// TIA Portal V19 export
FUNCTION "SUBOUTPUT" : Void   // FC4, LAD
{ S7_Optimized_Access := 'TRUE' }
// stored: SetENOAutomatically false
BEGIN

REGION Network 1: P-202 A RO 1 FEED PUMP
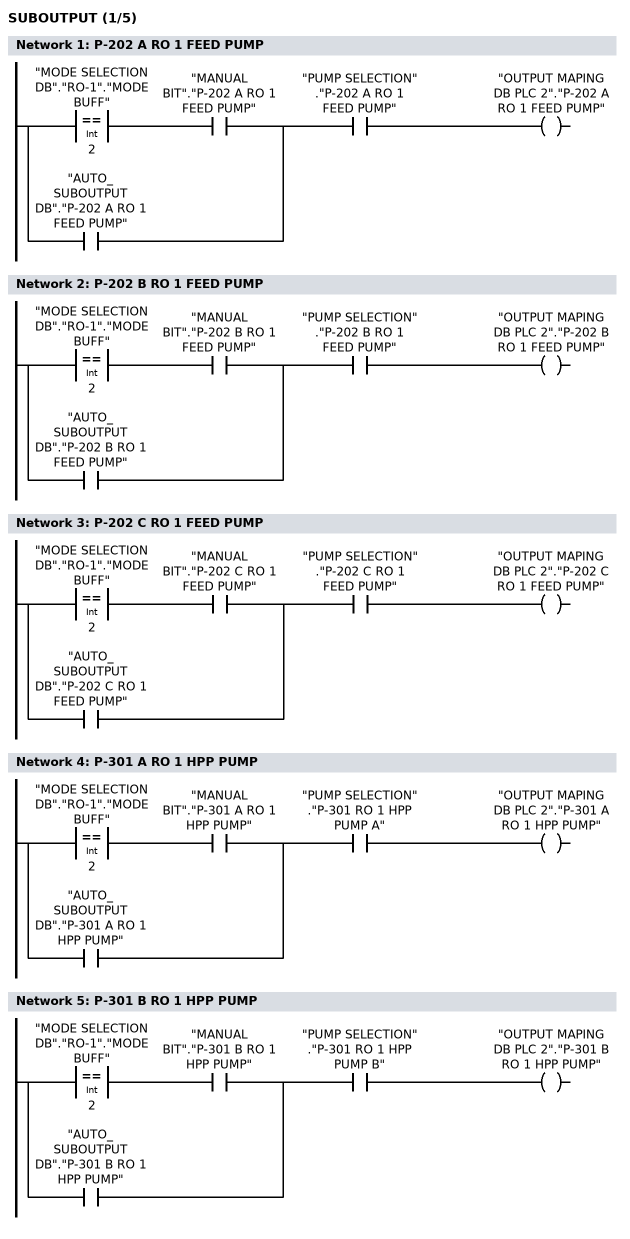
   RUNG wire#powerrail
      { S7_Templates := "SrcType := Int" } EQ_Contact(in1 := "MODE SELECTION DB"."RO-1"."MODE BUFF", in2 := 2)
      Contact( "MANUAL BIT"."P-202 A RO 1 FEED PUMP" )
      wire#w1
      Contact( "PUMP SELECTION"."P-202 A RO 1 FEED PUMP" )
      Coil( "OUTPUT MAPING DB PLC 2"."P-202 A RO 1 FEED PUMP" )
   END_RUNG
   RUNG wire#powerrail
      Contact( "AUTO_SUBOUTPUT DB"."P-202 A RO 1 FEED PUMP" )
   END_RUNG wire#w1
   // the same network as SCL:
   "OUTPUT MAPING DB PLC 2"."P-202 A RO 1 FEED PUMP" := ((("MODE SELECTION DB"."RO-1"."MODE BUFF" = 2) AND "MANUAL BIT"."P-202 A RO 1 FEED PUMP") OR "AUTO_SUBOUTPUT DB"."P-202 A RO 1 FEED PUMP") AND "PUMP SELECTION"."P-202 A RO 1 FEED PUMP";
END_REGION

REGION Network 2: P-202 B RO 1 FEED PUMP
   RUNG wire#powerrail
      { S7_Templates := "SrcType := Int" } EQ_Contact(in1 := "MODE SELECTION DB"."RO-1"."MODE BUFF", in2 := 2)
      Contact( "MANUAL BIT"."P-202 B RO 1 FEED PUMP" )
      wire#w1
      Contact( "PUMP SELECTION"."P-202 B RO 1 FEED PUMP" )
      Coil( "OUTPUT MAPING DB PLC 2"."P-202 B RO 1 FEED PUMP" )
   END_RUNG
   RUNG wire#powerrail
      Contact( "AUTO_SUBOUTPUT DB"."P-202 B RO 1 FEED PUMP" )
   END_RUNG wire#w1
   // the same network as SCL:
   "OUTPUT MAPING DB PLC 2"."P-202 B RO 1 FEED PUMP" := ((("MODE SELECTION DB"."RO-1"."MODE BUFF" = 2) AND "MANUAL BIT"."P-202 B RO 1 FEED PUMP") OR "AUTO_SUBOUTPUT DB"."P-202 B RO 1 FEED PUMP") AND "PUMP SELECTION"."P-202 B RO 1 FEED PUMP";
END_REGION

REGION Network 3: P-202 C RO 1 FEED PUMP
   RUNG wire#powerrail
      { S7_Templates := "SrcType := Int" } EQ_Contact(in1 := "MODE SELECTION DB"."RO-1"."MODE BUFF", in2 := 2)
      Contact( "MANUAL BIT"."P-202 C RO 1 FEED PUMP" )
      wire#w1
      Contact( "PUMP SELECTION"."P-202 C RO 1 FEED PUMP" )
      Coil( "OUTPUT MAPING DB PLC 2"."P-202 C RO 1 FEED PUMP" )
   END_RUNG
   RUNG wire#powerrail
      Contact( "AUTO_SUBOUTPUT DB"."P-202 C RO 1 FEED PUMP" )
   END_RUNG wire#w1
   // the same network as SCL:
   "OUTPUT MAPING DB PLC 2"."P-202 C RO 1 FEED PUMP" := ((("MODE SELECTION DB"."RO-1"."MODE BUFF" = 2) AND "MANUAL BIT"."P-202 C RO 1 FEED PUMP") OR "AUTO_SUBOUTPUT DB"."P-202 C RO 1 FEED PUMP") AND "PUMP SELECTION"."P-202 C RO 1 FEED PUMP";
END_REGION

REGION Network 4: P-301 A RO 1 HPP PUMP
   RUNG wire#powerrail
      { S7_Templates := "SrcType := Int" } EQ_Contact(in1 := "MODE SELECTION DB"."RO-1"."MODE BUFF", in2 := 2)
      Contact( "MANUAL BIT"."P-301 A RO 1 HPP PUMP" )
      wire#w1
      Contact( "PUMP SELECTION"."P-301 RO 1 HPP PUMP A" )
      Coil( "OUTPUT MAPING DB PLC 2"."P-301 A RO 1 HPP PUMP" )
   END_RUNG
   RUNG wire#powerrail
      Contact( "AUTO_SUBOUTPUT DB"."P-301 A RO 1 HPP PUMP" )
   END_RUNG wire#w1
   // the same network as SCL:
   "OUTPUT MAPING DB PLC 2"."P-301 A RO 1 HPP PUMP" := ((("MODE SELECTION DB"."RO-1"."MODE BUFF" = 2) AND "MANUAL BIT"."P-301 A RO 1 HPP PUMP") OR "AUTO_SUBOUTPUT DB"."P-301 A RO 1 HPP PUMP") AND "PUMP SELECTION"."P-301 RO 1 HPP PUMP A";
END_REGION

REGION Network 5: P-301 B RO 1 HPP PUMP
   RUNG wire#powerrail
      { S7_Templates := "SrcType := Int" } EQ_Contact(in1 := "MODE SELECTION DB"."RO-1"."MODE BUFF", in2 := 2)
      Contact( "MANUAL BIT"."P-301 B RO 1 HPP PUMP" )
      wire#w1
      Contact( "PUMP SELECTION"."P-301 RO 1 HPP PUMP B" )
      Coil( "OUTPUT MAPING DB PLC 2"."P-301 B RO 1 HPP PUMP" )
   END_RUNG
   RUNG wire#powerrail
      Contact( "AUTO_SUBOUTPUT DB"."P-301 B RO 1 HPP PUMP" )
   END_RUNG wire#w1
   // the same network as SCL:
   "OUTPUT MAPING DB PLC 2"."P-301 B RO 1 HPP PUMP" := ((("MODE SELECTION DB"."RO-1"."MODE BUFF" = 2) AND "MANUAL BIT"."P-301 B RO 1 HPP PUMP") OR "AUTO_SUBOUTPUT DB"."P-301 B RO 1 HPP PUMP") AND "PUMP SELECTION"."P-301 RO 1 HPP PUMP B";
END_REGION

REGION Network 6: P-401 A RO 2 FEED PUMP
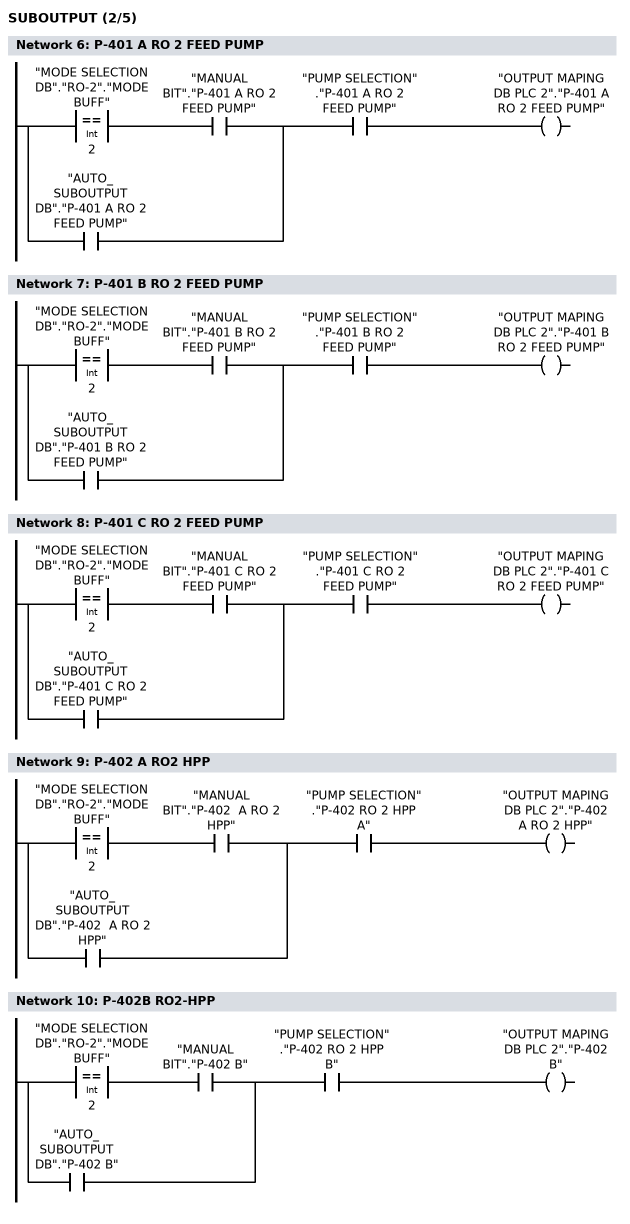
   RUNG wire#powerrail
      { S7_Templates := "SrcType := Int" } EQ_Contact(in1 := "MODE SELECTION DB"."RO-2"."MODE BUFF", in2 := 2)
      Contact( "MANUAL BIT"."P-401 A RO 2 FEED PUMP" )
      wire#w1
      Contact( "PUMP SELECTION"."P-401 A RO 2 FEED PUMP" )
      Coil( "OUTPUT MAPING DB PLC 2"."P-401 A RO 2 FEED PUMP" )
   END_RUNG
   RUNG wire#powerrail
      Contact( "AUTO_SUBOUTPUT DB"."P-401 A RO 2 FEED PUMP" )
   END_RUNG wire#w1
   // the same network as SCL:
   "OUTPUT MAPING DB PLC 2"."P-401 A RO 2 FEED PUMP" := ((("MODE SELECTION DB"."RO-2"."MODE BUFF" = 2) AND "MANUAL BIT"."P-401 A RO 2 FEED PUMP") OR "AUTO_SUBOUTPUT DB"."P-401 A RO 2 FEED PUMP") AND "PUMP SELECTION"."P-401 A RO 2 FEED PUMP";
END_REGION

REGION Network 7: P-401 B RO 2 FEED PUMP
   RUNG wire#powerrail
      { S7_Templates := "SrcType := Int" } EQ_Contact(in1 := "MODE SELECTION DB"."RO-2"."MODE BUFF", in2 := 2)
      Contact( "MANUAL BIT"."P-401 B RO 2 FEED PUMP" )
      wire#w1
      Contact( "PUMP SELECTION"."P-401 B RO 2 FEED PUMP" )
      Coil( "OUTPUT MAPING DB PLC 2"."P-401 B RO 2 FEED PUMP" )
   END_RUNG
   RUNG wire#powerrail
      Contact( "AUTO_SUBOUTPUT DB"."P-401 B RO 2 FEED PUMP" )
   END_RUNG wire#w1
   // the same network as SCL:
   "OUTPUT MAPING DB PLC 2"."P-401 B RO 2 FEED PUMP" := ((("MODE SELECTION DB"."RO-2"."MODE BUFF" = 2) AND "MANUAL BIT"."P-401 B RO 2 FEED PUMP") OR "AUTO_SUBOUTPUT DB"."P-401 B RO 2 FEED PUMP") AND "PUMP SELECTION"."P-401 B RO 2 FEED PUMP";
END_REGION

REGION Network 8: P-401 C RO 2 FEED PUMP
   RUNG wire#powerrail
      { S7_Templates := "SrcType := Int" } EQ_Contact(in1 := "MODE SELECTION DB"."RO-2"."MODE BUFF", in2 := 2)
      Contact( "MANUAL BIT"."P-401 C RO 2 FEED PUMP" )
      wire#w1
      Contact( "PUMP SELECTION"."P-401 C RO 2 FEED PUMP" )
      Coil( "OUTPUT MAPING DB PLC 2"."P-401 C RO 2 FEED PUMP" )
   END_RUNG
   RUNG wire#powerrail
      Contact( "AUTO_SUBOUTPUT DB"."P-401 C RO 2 FEED PUMP" )
   END_RUNG wire#w1
   // the same network as SCL:
   "OUTPUT MAPING DB PLC 2"."P-401 C RO 2 FEED PUMP" := ((("MODE SELECTION DB"."RO-2"."MODE BUFF" = 2) AND "MANUAL BIT"."P-401 C RO 2 FEED PUMP") OR "AUTO_SUBOUTPUT DB"."P-401 C RO 2 FEED PUMP") AND "PUMP SELECTION"."P-401 C RO 2 FEED PUMP";
END_REGION

REGION Network 9: P-402 A RO2 HPP
   RUNG wire#powerrail
      { S7_Templates := "SrcType := Int" } EQ_Contact(in1 := "MODE SELECTION DB"."RO-2"."MODE BUFF", in2 := 2)
      Contact( "MANUAL BIT"."P-402  A RO 2 HPP" )
      wire#w1
      Contact( "PUMP SELECTION"."P-402 RO 2 HPP A" )
      Coil( "OUTPUT MAPING DB PLC 2"."P-402  A RO 2 HPP" )
   END_RUNG
   RUNG wire#powerrail
      Contact( "AUTO_SUBOUTPUT DB"."P-402  A RO 2 HPP" )
   END_RUNG wire#w1
   // the same network as SCL:
   "OUTPUT MAPING DB PLC 2"."P-402  A RO 2 HPP" := ((("MODE SELECTION DB"."RO-2"."MODE BUFF" = 2) AND "MANUAL BIT"."P-402  A RO 2 HPP") OR "AUTO_SUBOUTPUT DB"."P-402  A RO 2 HPP") AND "PUMP SELECTION"."P-402 RO 2 HPP A";
END_REGION

REGION Network 10: P-402B RO2-HPP
   RUNG wire#powerrail
      { S7_Templates := "SrcType := Int" } EQ_Contact(in1 := "MODE SELECTION DB"."RO-2"."MODE BUFF", in2 := 2)
      Contact( "MANUAL BIT"."P-402 B" )
      wire#w1
      Contact( "PUMP SELECTION"."P-402 RO 2 HPP B" )
      Coil( "OUTPUT MAPING DB PLC 2"."P-402 B" )
   END_RUNG
   RUNG wire#powerrail
      Contact( "AUTO_SUBOUTPUT DB"."P-402 B" )
   END_RUNG wire#w1
   // the same network as SCL:
   "OUTPUT MAPING DB PLC 2"."P-402 B" := ((("MODE SELECTION DB"."RO-2"."MODE BUFF" = 2) AND "MANUAL BIT"."P-402 B") OR "AUTO_SUBOUTPUT DB"."P-402 B") AND "PUMP SELECTION"."P-402 RO 2 HPP B";
END_REGION

REGION Network 11: P-501 A EDI FEED PUMP
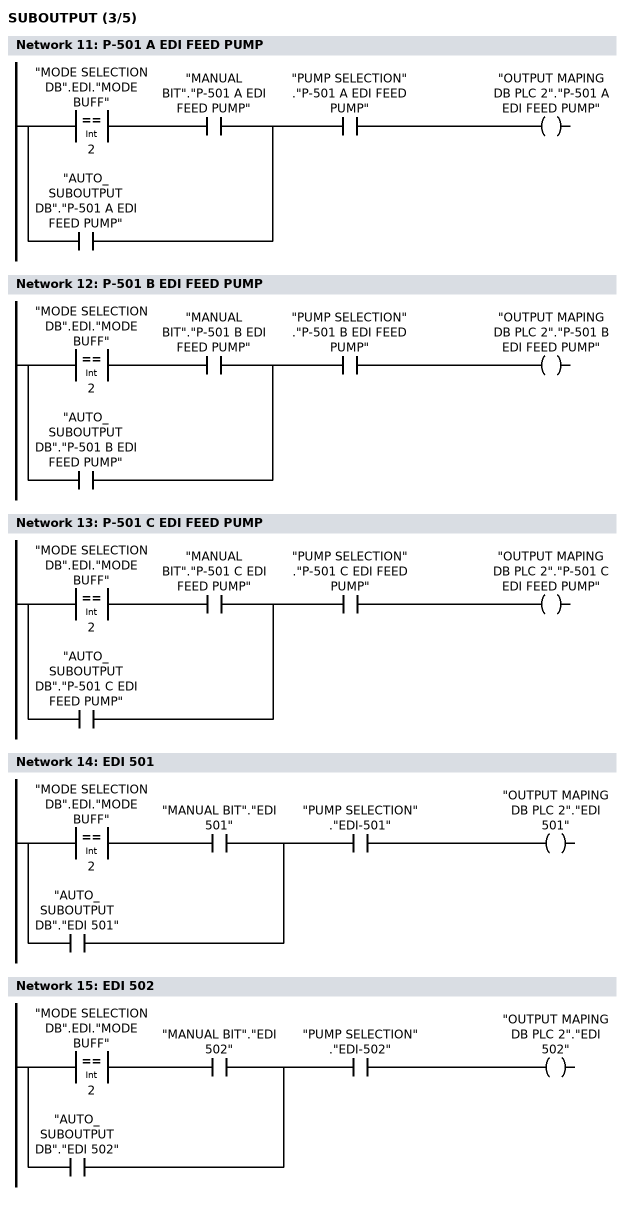
   RUNG wire#powerrail
      { S7_Templates := "SrcType := Int" } EQ_Contact(in1 := "MODE SELECTION DB".EDI."MODE BUFF", in2 := 2)
      Contact( "MANUAL BIT"."P-501 A EDI FEED PUMP" )
      wire#w1
      Contact( "PUMP SELECTION"."P-501 A EDI FEED PUMP" )
      Coil( "OUTPUT MAPING DB PLC 2"."P-501 A EDI FEED PUMP" )
   END_RUNG
   RUNG wire#powerrail
      Contact( "AUTO_SUBOUTPUT DB"."P-501 A EDI FEED PUMP" )
   END_RUNG wire#w1
   // the same network as SCL:
   "OUTPUT MAPING DB PLC 2"."P-501 A EDI FEED PUMP" := ((("MODE SELECTION DB".EDI."MODE BUFF" = 2) AND "MANUAL BIT"."P-501 A EDI FEED PUMP") OR "AUTO_SUBOUTPUT DB"."P-501 A EDI FEED PUMP") AND "PUMP SELECTION"."P-501 A EDI FEED PUMP";
END_REGION

REGION Network 12: P-501 B EDI FEED PUMP
   RUNG wire#powerrail
      { S7_Templates := "SrcType := Int" } EQ_Contact(in1 := "MODE SELECTION DB".EDI."MODE BUFF", in2 := 2)
      Contact( "MANUAL BIT"."P-501 B EDI FEED PUMP" )
      wire#w1
      Contact( "PUMP SELECTION"."P-501 B EDI FEED PUMP" )
      Coil( "OUTPUT MAPING DB PLC 2"."P-501 B EDI FEED PUMP" )
   END_RUNG
   RUNG wire#powerrail
      Contact( "AUTO_SUBOUTPUT DB"."P-501 B EDI FEED PUMP" )
   END_RUNG wire#w1
   // the same network as SCL:
   "OUTPUT MAPING DB PLC 2"."P-501 B EDI FEED PUMP" := ((("MODE SELECTION DB".EDI."MODE BUFF" = 2) AND "MANUAL BIT"."P-501 B EDI FEED PUMP") OR "AUTO_SUBOUTPUT DB"."P-501 B EDI FEED PUMP") AND "PUMP SELECTION"."P-501 B EDI FEED PUMP";
END_REGION

REGION Network 13: P-501 C EDI FEED PUMP
   RUNG wire#powerrail
      { S7_Templates := "SrcType := Int" } EQ_Contact(in1 := "MODE SELECTION DB".EDI."MODE BUFF", in2 := 2)
      Contact( "MANUAL BIT"."P-501 C EDI FEED PUMP" )
      wire#w1
      Contact( "PUMP SELECTION"."P-501 C EDI FEED PUMP" )
      Coil( "OUTPUT MAPING DB PLC 2"."P-501 C EDI FEED PUMP" )
   END_RUNG
   RUNG wire#powerrail
      Contact( "AUTO_SUBOUTPUT DB"."P-501 C EDI FEED PUMP" )
   END_RUNG wire#w1
   // the same network as SCL:
   "OUTPUT MAPING DB PLC 2"."P-501 C EDI FEED PUMP" := ((("MODE SELECTION DB".EDI."MODE BUFF" = 2) AND "MANUAL BIT"."P-501 C EDI FEED PUMP") OR "AUTO_SUBOUTPUT DB"."P-501 C EDI FEED PUMP") AND "PUMP SELECTION"."P-501 C EDI FEED PUMP";
END_REGION

REGION Network 14: EDI 501
   RUNG wire#powerrail
      { S7_Templates := "SrcType := Int" } EQ_Contact(in1 := "MODE SELECTION DB".EDI."MODE BUFF", in2 := 2)
      Contact( "MANUAL BIT"."EDI 501" )
      wire#w1
      Contact( "PUMP SELECTION"."EDI-501" )
      Coil( "OUTPUT MAPING DB PLC 2"."EDI 501" )
   END_RUNG
   RUNG wire#powerrail
      Contact( "AUTO_SUBOUTPUT DB"."EDI 501" )
   END_RUNG wire#w1
   // the same network as SCL:
   "OUTPUT MAPING DB PLC 2"."EDI 501" := ((("MODE SELECTION DB".EDI."MODE BUFF" = 2) AND "MANUAL BIT"."EDI 501") OR "AUTO_SUBOUTPUT DB"."EDI 501") AND "PUMP SELECTION"."EDI-501";
END_REGION

REGION Network 15: EDI 502
   RUNG wire#powerrail
      { S7_Templates := "SrcType := Int" } EQ_Contact(in1 := "MODE SELECTION DB".EDI."MODE BUFF", in2 := 2)
      Contact( "MANUAL BIT"."EDI 502" )
      wire#w1
      Contact( "PUMP SELECTION"."EDI-502" )
      Coil( "OUTPUT MAPING DB PLC 2"."EDI 502" )
   END_RUNG
   RUNG wire#powerrail
      Contact( "AUTO_SUBOUTPUT DB"."EDI 502" )
   END_RUNG wire#w1
   // the same network as SCL:
   "OUTPUT MAPING DB PLC 2"."EDI 502" := ((("MODE SELECTION DB".EDI."MODE BUFF" = 2) AND "MANUAL BIT"."EDI 502") OR "AUTO_SUBOUTPUT DB"."EDI 502") AND "PUMP SELECTION"."EDI-502";
END_REGION

REGION Network 16: DP 703
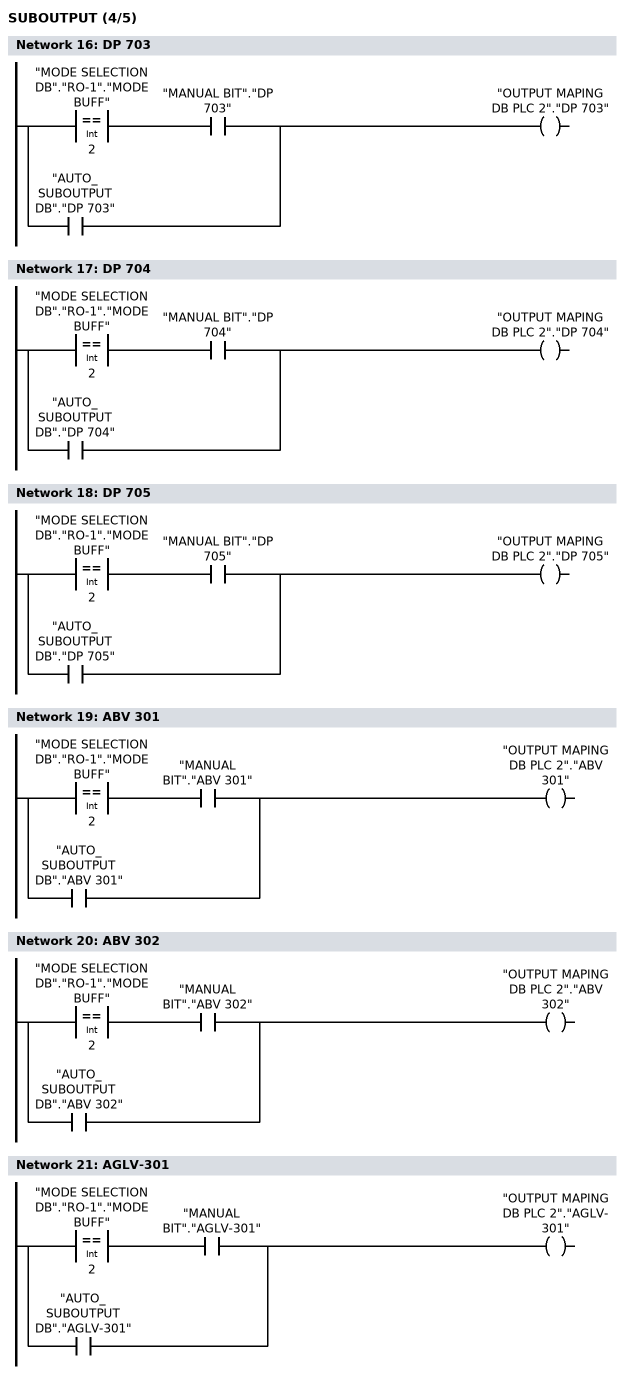
   RUNG wire#powerrail
      { S7_Templates := "SrcType := Int" } EQ_Contact(in1 := "MODE SELECTION DB"."RO-1"."MODE BUFF", in2 := 2)
      Contact( "MANUAL BIT"."DP 703" )
      wire#w1
      Coil( "OUTPUT MAPING DB PLC 2"."DP 703" )
   END_RUNG
   RUNG wire#powerrail
      Contact( "AUTO_SUBOUTPUT DB"."DP 703" )
   END_RUNG wire#w1
   // the same network as SCL:
   "OUTPUT MAPING DB PLC 2"."DP 703" := (("MODE SELECTION DB"."RO-1"."MODE BUFF" = 2) AND "MANUAL BIT"."DP 703") OR "AUTO_SUBOUTPUT DB"."DP 703";
END_REGION

REGION Network 17: DP 704
   RUNG wire#powerrail
      { S7_Templates := "SrcType := Int" } EQ_Contact(in1 := "MODE SELECTION DB"."RO-1"."MODE BUFF", in2 := 2)
      Contact( "MANUAL BIT"."DP 704" )
      wire#w1
      Coil( "OUTPUT MAPING DB PLC 2"."DP 704" )
   END_RUNG
   RUNG wire#powerrail
      Contact( "AUTO_SUBOUTPUT DB"."DP 704" )
   END_RUNG wire#w1
   // the same network as SCL:
   "OUTPUT MAPING DB PLC 2"."DP 704" := (("MODE SELECTION DB"."RO-1"."MODE BUFF" = 2) AND "MANUAL BIT"."DP 704") OR "AUTO_SUBOUTPUT DB"."DP 704";
END_REGION

REGION Network 18: DP 705
   RUNG wire#powerrail
      { S7_Templates := "SrcType := Int" } EQ_Contact(in1 := "MODE SELECTION DB"."RO-1"."MODE BUFF", in2 := 2)
      Contact( "MANUAL BIT"."DP 705" )
      wire#w1
      Coil( "OUTPUT MAPING DB PLC 2"."DP 705" )
   END_RUNG
   RUNG wire#powerrail
      Contact( "AUTO_SUBOUTPUT DB"."DP 705" )
   END_RUNG wire#w1
   // the same network as SCL:
   "OUTPUT MAPING DB PLC 2"."DP 705" := (("MODE SELECTION DB"."RO-1"."MODE BUFF" = 2) AND "MANUAL BIT"."DP 705") OR "AUTO_SUBOUTPUT DB"."DP 705";
END_REGION

REGION Network 19: ABV 301
   RUNG wire#powerrail
      { S7_Templates := "SrcType := Int" } EQ_Contact(in1 := "MODE SELECTION DB"."RO-1"."MODE BUFF", in2 := 2)
      Contact( "MANUAL BIT"."ABV 301" )
      wire#w1
      Coil( "OUTPUT MAPING DB PLC 2"."ABV 301" )
   END_RUNG
   RUNG wire#powerrail
      Contact( "AUTO_SUBOUTPUT DB"."ABV 301" )
   END_RUNG wire#w1
   // the same network as SCL:
   "OUTPUT MAPING DB PLC 2"."ABV 301" := (("MODE SELECTION DB"."RO-1"."MODE BUFF" = 2) AND "MANUAL BIT"."ABV 301") OR "AUTO_SUBOUTPUT DB"."ABV 301";
END_REGION

REGION Network 20: ABV 302
   RUNG wire#powerrail
      { S7_Templates := "SrcType := Int" } EQ_Contact(in1 := "MODE SELECTION DB"."RO-1"."MODE BUFF", in2 := 2)
      Contact( "MANUAL BIT"."ABV 302" )
      wire#w1
      Coil( "OUTPUT MAPING DB PLC 2"."ABV 302" )
   END_RUNG
   RUNG wire#powerrail
      Contact( "AUTO_SUBOUTPUT DB"."ABV 302" )
   END_RUNG wire#w1
   // the same network as SCL:
   "OUTPUT MAPING DB PLC 2"."ABV 302" := (("MODE SELECTION DB"."RO-1"."MODE BUFF" = 2) AND "MANUAL BIT"."ABV 302") OR "AUTO_SUBOUTPUT DB"."ABV 302";
END_REGION

REGION Network 21: AGLV-301
   RUNG wire#powerrail
      { S7_Templates := "SrcType := Int" } EQ_Contact(in1 := "MODE SELECTION DB"."RO-1"."MODE BUFF", in2 := 2)
      Contact( "MANUAL BIT"."AGLV-301" )
      wire#w1
      Coil( "OUTPUT MAPING DB PLC 2"."AGLV-301" )
   END_RUNG
   RUNG wire#powerrail
      Contact( "AUTO_SUBOUTPUT DB"."AGLV-301" )
   END_RUNG wire#w1
   // the same network as SCL:
   "OUTPUT MAPING DB PLC 2"."AGLV-301" := (("MODE SELECTION DB"."RO-1"."MODE BUFF" = 2) AND "MANUAL BIT"."AGLV-301") OR "AUTO_SUBOUTPUT DB"."AGLV-301";
END_REGION

REGION Network 22: AGLV-302
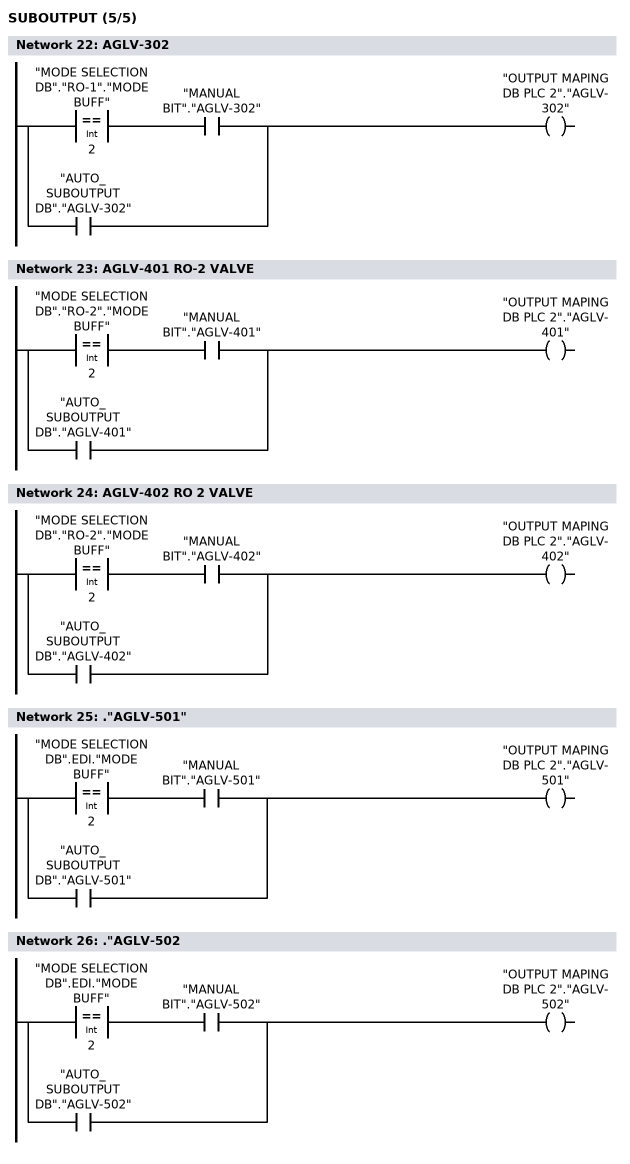
   RUNG wire#powerrail
      { S7_Templates := "SrcType := Int" } EQ_Contact(in1 := "MODE SELECTION DB"."RO-1"."MODE BUFF", in2 := 2)
      Contact( "MANUAL BIT"."AGLV-302" )
      wire#w1
      Coil( "OUTPUT MAPING DB PLC 2"."AGLV-302" )
   END_RUNG
   RUNG wire#powerrail
      Contact( "AUTO_SUBOUTPUT DB"."AGLV-302" )
   END_RUNG wire#w1
   // the same network as SCL:
   "OUTPUT MAPING DB PLC 2"."AGLV-302" := (("MODE SELECTION DB"."RO-1"."MODE BUFF" = 2) AND "MANUAL BIT"."AGLV-302") OR "AUTO_SUBOUTPUT DB"."AGLV-302";
END_REGION

REGION Network 23: AGLV-401 RO-2 VALVE
   RUNG wire#powerrail
      { S7_Templates := "SrcType := Int" } EQ_Contact(in1 := "MODE SELECTION DB"."RO-2"."MODE BUFF", in2 := 2)
      Contact( "MANUAL BIT"."AGLV-401" )
      wire#w1
      Coil( "OUTPUT MAPING DB PLC 2"."AGLV-401" )
   END_RUNG
   RUNG wire#powerrail
      Contact( "AUTO_SUBOUTPUT DB"."AGLV-401" )
   END_RUNG wire#w1
   // the same network as SCL:
   "OUTPUT MAPING DB PLC 2"."AGLV-401" := (("MODE SELECTION DB"."RO-2"."MODE BUFF" = 2) AND "MANUAL BIT"."AGLV-401") OR "AUTO_SUBOUTPUT DB"."AGLV-401";
END_REGION

REGION Network 24: AGLV-402 RO 2 VALVE
   RUNG wire#powerrail
      { S7_Templates := "SrcType := Int" } EQ_Contact(in1 := "MODE SELECTION DB"."RO-2"."MODE BUFF", in2 := 2)
      Contact( "MANUAL BIT"."AGLV-402" )
      wire#w1
      Coil( "OUTPUT MAPING DB PLC 2"."AGLV-402" )
   END_RUNG
   RUNG wire#powerrail
      Contact( "AUTO_SUBOUTPUT DB"."AGLV-402" )
   END_RUNG wire#w1
   // the same network as SCL:
   "OUTPUT MAPING DB PLC 2"."AGLV-402" := (("MODE SELECTION DB"."RO-2"."MODE BUFF" = 2) AND "MANUAL BIT"."AGLV-402") OR "AUTO_SUBOUTPUT DB"."AGLV-402";
END_REGION

REGION Network 25: ."AGLV-501"
   RUNG wire#powerrail
      { S7_Templates := "SrcType := Int" } EQ_Contact(in1 := "MODE SELECTION DB".EDI."MODE BUFF", in2 := 2)
      Contact( "MANUAL BIT"."AGLV-501" )
      wire#w1
      Coil( "OUTPUT MAPING DB PLC 2"."AGLV-501" )
   END_RUNG
   RUNG wire#powerrail
      Contact( "AUTO_SUBOUTPUT DB"."AGLV-501" )
   END_RUNG wire#w1
   // the same network as SCL:
   "OUTPUT MAPING DB PLC 2"."AGLV-501" := (("MODE SELECTION DB".EDI."MODE BUFF" = 2) AND "MANUAL BIT"."AGLV-501") OR "AUTO_SUBOUTPUT DB"."AGLV-501";
END_REGION

REGION Network 26: ."AGLV-502
   RUNG wire#powerrail
      { S7_Templates := "SrcType := Int" } EQ_Contact(in1 := "MODE SELECTION DB".EDI."MODE BUFF", in2 := 2)
      Contact( "MANUAL BIT"."AGLV-502" )
      wire#w1
      Coil( "OUTPUT MAPING DB PLC 2"."AGLV-502" )
   END_RUNG
   RUNG wire#powerrail
      Contact( "AUTO_SUBOUTPUT DB"."AGLV-502" )
   END_RUNG wire#w1
   // the same network as SCL:
   "OUTPUT MAPING DB PLC 2"."AGLV-502" := (("MODE SELECTION DB".EDI."MODE BUFF" = 2) AND "MANUAL BIT"."AGLV-502") OR "AUTO_SUBOUTPUT DB"."AGLV-502";
END_REGION
END_FUNCTION
